FUNCTION_BLOCK RandomEvent (* Composite Function Block Type *)
  (* Standard: 61499-2 *)
  (* Version 0.0, 8/30/2016, Dmitry, nxtControl GmbH, template *)
  PACKAGE Main;
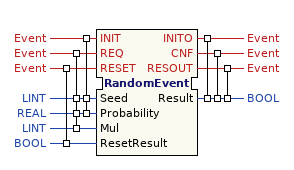
  EVENT_INPUT
    INIT WITH Seed, Probability; (* Initialization Request *)
    REQ WITH Seed, Probability, Mul; (* Normal Execution Request *)
    RESET WITH ResetResult;
  END_EVENT
  EVENT_OUTPUT
    INITO WITH Result; (* Initialization Confirm *)
    CNF WITH Result; (* Execution Confirmation *)
    RESOUT WITH Result;
  END_EVENT
  VAR_INPUT
    Seed : LINT;
    Probability : REAL;
    Mul : LINT;
    ResetResult : BOOL;
  END_VAR
  VAR_OUTPUT
    Result : BOOL;
  END_VAR
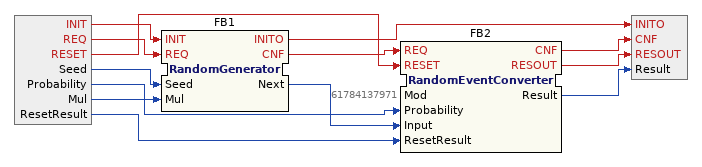
  FBS
    FB1 : RandomGenerator;
    FB2 : RandomEventConverter(Mod := 61784137971);
  END_FBS
  EVENT_CONNECTIONS
    INIT TO FB1.INIT;
    REQ TO FB1.REQ;
    FB1.INITO TO INITO;
    FB2.CNF TO CNF;
    FB1.CNF TO FB2.REQ;
    RESET TO FB2.RESET;
    FB2.RESOUT TO RESOUT;
  END_CONNECTIONS
  DATA_CONNECTIONS
    Seed TO FB1.Seed;
    FB1.Next TO FB2.Input;
    Probability TO FB2.Probability;
    FB2.Result TO Result;
    Mul TO FB1.Mul;
    ResetResult TO FB2.ResetResult;
  END_CONNECTIONS
END_FUNCTION_BLOCK
